// TwinCAT 3 PLC project StageUtils
// Title: StageUtils
// Company: _
// Author: Krystian Lis et al.
// ProjectVersion: 2.0.0
// Description: Various Stage related utilities
// ProgramVersion: 3.1.4026.16
// libraries:
//   Tc2_Standard, * (Beckhoff Automation GmbH)
//   Tc2_System, * (Beckhoff Automation GmbH)
//   StageCore, * (_)
// project tree:
//   Arg/ArgList/ ArgList.TcPOU, I_ArgList.TcIO (not stored), I_MutArgList.TcIO
//   Arg/ArgQueue/ ArgQueue.TcPOU, I_ArgQueue.TcIO, I_MutArgQueue.TcIO
//   Color/ Color.TcDUT, RgbColor.TcPOU
//   Color/Itf/ I_RgbColor.TcIO
//   Entity/CompList/ CompList.TcPOU, I_CompList.TcIO (not stored), I_MutCompList.TcIO
//   Entity/CompSet/ CompSet.TcPOU, I_CompSet.TcIO
//   Math/ Math.TcPOU
//   Time/ GetTaskCycleTime.TcPOU (not stored), GetUnixTime.TcPOU (not stored)
// real-time tasks:
//   TASK Example: cycle T#10ms, priority 20, ADS port 350
//   TASK Test: cycle T#10ms, priority 21, ADS port 351
//   TASK VISU_TASK: cycle T#200000us, priority 30, ADS port 352

// ---- Color/Color.TcDUT
(*
A DWORD alias type to be used with PLC HMI. Encodes RGB value.
*)
TYPE Color : DWORD; END_TYPE

// ---- Arg/ArgList/I_MutArgList.TcIO
(*
A list implementation for managing `I_Arg`.  
*)
INTERFACE I_MutArgList EXTENDS I_ArgList

(*
Adds, updates, or removes an argument in the list at the specified index.  
Return:
- `Ok` - Upon successfully adding, modifying, or removing an entry.
- `Err.Idx` - When attempting to modify an entry at an out-of-bounds index.
*)
METHOD Set : Result
VAR_INPUT
	iIn		: I_Arg;
	nIndex		: UDINT;
END_VAR
END_METHOD

END_INTERFACE

// ---- Arg/ArgQueue/I_ArgQueue.TcIO
(*
A circular queue implementation for managing `I_Arg`.  
*)
INTERFACE I_ArgQueue EXTENDS I_Debug

(*
Returns the current head index of the queue, indicating the next position for insertion.
*)
PROPERTY Head : UDINT
GET
END_GET
END_PROPERTY

PROPERTY Length : UDINT
GET
END_GET
END_PROPERTY

(*
Provides access to the underlying list structure that holds the queue's argument objects.
*)
PROPERTY List : I_ArgList
GET
END_GET
END_PROPERTY

(*
Returns the current tail index of the queue, indicating the next position for retrieval.
*)
PROPERTY Tail : UDINT
GET
END_GET
END_PROPERTY

END_INTERFACE

// ---- Arg/ArgQueue/I_MutArgQueue.TcIO
(*
A circular queue implementation for managing `I_Arg`.  
*)
INTERFACE I_MutArgQueue EXTENDS I_ArgQueue

(*
Clears the queue.
*)
METHOD Clear
END_METHOD

(*
Retrieves and removes the next argument from the queue.  
Advances the tail pointer, ensuring cyclic operation within the queue's capacity.
Returns:
- Ok - Returns `I_Arg`.
- Err.NotFound - Returns null, queue empty.
- Check `I_MutArgList.Get` for more results.
*)
METHOD Pop : Result
VAR_INPUT
	iOut	: REFERENCE TO I_Arg;
END_VAR
END_METHOD

(*
Adds a new argument to the queue.  
Advances the head pointer while maintaining a cyclic structure, and returns an overflow error if the queue is full.
Returns:
- Ok - Successful insertion.
- Err.Ovf - Returns null, the queue is full.
- Check `I_MutArgList.Set` for more results.
*)
METHOD Push : Result
VAR_INPUT
	iIn		: I_Arg;
END_VAR
END_METHOD

END_INTERFACE

// ---- Color/Itf/I_RgbColor.TcIO
(*
Provides methods and properties to operate on RGBA value.
*)
INTERFACE I_RgbColor

(*
ALPHA channel
*)
PROPERTY Alpha : BYTE
GET
END_GET
SET
END_SET
END_PROPERTY

(*
BLUE component
*)
PROPERTY Blue : BYTE
GET
END_GET
SET
END_SET
END_PROPERTY

(*
Clones other components of I_RgbaColor interface.
*)
METHOD Clone
VAR_INPUT
	iColor	: I_RgbColor;
END_VAR
END_METHOD

(*
GREEN component
*)
PROPERTY Green : BYTE
GET
END_GET
SET
END_SET
END_PROPERTY

(*
Compute single Color value from RGBA components when used as getter.
Sets RGBA values by extracting components from a single Color value.
*)
PROPERTY Raw : Color
GET
END_GET
SET
END_SET
END_PROPERTY

(*
RED component
*)
PROPERTY Red : BYTE
GET
END_GET
SET
END_SET
END_PROPERTY

(*
Set each RGBA component value separately.
*)
METHOD Set
VAR_INPUT
	nRed: USINT;
	nGreen: USINT;
	nBlue: USINT;
	nAlpha: USINT;
END_VAR
END_METHOD

END_INTERFACE

// ---- Entity/CompList/I_MutCompList.TcIO
(*
A list implementation for managing `I_Component`.  
*)
INTERFACE I_MutCompList EXTENDS I_CompList

(*
Adds, updates, or removes an argument in the list at the specified index.  
Return:
- `Ok` - Upon successfully adding, modifying, or removing an entry.
- `Err.Idx` - When attempting to modify an entry at an out-of-bounds index.
*)
METHOD Set : Result
VAR_INPUT
	iIn			: I_Component;
	nIndex		: UDINT;
END_VAR
END_METHOD

END_INTERFACE

// ---- Entity/CompSet/I_CompSet.TcIO
INTERFACE I_CompSet

METHOD Append : Result
VAR_INPUT
	iComp: I_Component;
END_VAR
END_METHOD

METHOD Get : Result
VAR_INPUT
	nIdx: UDINT;
	iResult: REFERENCE TO I_Component;
END_VAR
END_METHOD

END_INTERFACE

// ---- Arg/ArgList/ArgList.TcPOU
(*
A list implementation for managing `I_Arg`.  
*)
FUNCTION_BLOCK ArgList
VAR_GENERIC CONSTANT
	nCap	: UDINT := 100;
END_VAR

IMPLEMENTS I_MutArgList

VAR
	_iList	: ARRAY[1..nCap] OF I_Arg;
END_VAR

(*
Provides the maximum capacity of the list.
*)
PROPERTY Cap : UDINT
GET
Cap := nCap;
END_GET
END_PROPERTY

(*
Retrieves the `I_Arg` at the specified index.  
Returns:
- `Ok` - Successfully retrieves the `I_Arg`.
- `Err.Idx` - The specified index is out of bounds.
- `Err.InvRef` - Invalid output reference.
- `Err.Idx` - `iOut` = 0.
*)
METHOD Get : Result
VAR_INPUT
	nIndex		: UDINT;
	iOut		: REFERENCE TO I_Arg;
END_VAR
IF nIndex > nCap OR nIndex = 0 THEN
	Get := Err.Idx;
	RETURN;	
END_IF

IF NOT __ISVALIDREF(iOut) THEN
	Get := Err.InvRef;
	RETURN;
END_IF

iOut := _iList[nIndex];
IF iOut <> 0 THEN
	Get := Ok;
ELSE
	Get := Err.NotFound;
END_IF
END_METHOD

(*
Adds, updates, or removes an argument in the list at the specified index.  
Return:
- `Ok` - Upon successfully adding, modifying, or removing an entry.
- `Err.Idx` - When attempting to modify an entry at an out-of-bounds index.
*)
METHOD Set : Result
VAR_INPUT
	iIn		: I_Arg;
	nIndex		: UDINT;
END_VAR
IF nIndex > nCap OR nIndex = 0 THEN
	Set := Err.Idx;
	RETURN;	
END_IF

_iList[nIndex] := iIn;
Set := Ok;
END_METHOD

END_FUNCTION_BLOCK

// ---- Arg/ArgQueue/ArgQueue.TcPOU
(*
A circular queue implementation for managing `I_Arg`.  
*)
FUNCTION_BLOCK ArgQueue
VAR_GENERIC CONSTANT
	nCap		: UDINT := 100;
END_VAR

IMPLEMENTS I_MutArgQueue

VAR
	_list		: ArgList<nCap>;
	_nLen		: UDINT := 0;
	_nHead		: UDINT := 1;
	_nTail		: UDINT := 1;
END_VAR

(*
Clears the queue.
*)
METHOD Clear
_nHead := 1;
_nTail := 1;
_nLen := 0;
_list.Set(0, 1);
END_METHOD

(*
Returns the current head index of the queue, indicating the next position for insertion.
*)
PROPERTY Head : UDINT
GET
Head := _nHead;
END_GET
END_PROPERTY

PROPERTY Length : UDINT
GET
Length := _nLen;
END_GET
END_PROPERTY

(*
Provides access to the underlying list structure that holds the queue's argument objects.
*)
PROPERTY List : I_ArgList
GET
List := _list;
END_GET
END_PROPERTY

(*
Allows initializing an external interface variable with an interface pointer to this instance within declaration block.
Example:
iQueue: I_MutArgQueue;
queue: ArgQueue := (MutProxy := iQueue);
Result: iQueue <> 0 
*)
PROPERTY MutProxy : REFERENCE TO I_MutArgQueue
SET
MutProxy := THIS^;
END_SET
END_PROPERTY

(*
Retrieves and removes the next argument from the queue.  
Advances the tail pointer, ensuring cyclic operation within the queue's capacity.
Returns:
- Ok - Returns `I_Arg`.
- Err.NotFound - Returns null, queue empty.
- Check `I_ArgList.Get` for more results.
*)
METHOD Pop : Result
VAR_INPUT
	iOut	: REFERENCE TO I_Arg;
END_VAR
IF _nLen = 0 THEN
	Pop := Err.NotFound;
	RETURN;
END_IF;

IF IsOk(_list.Get(_nHead, iOut), nOut => Pop) THEN
	_nHead := (_nHead MOD nCap) + 1;
	_nLen := _nLen - 1;
	Pop := Ok;
END_IF;
END_METHOD

(*
Allows initializing an external interface variable with an interface pointer to this instance within declaration block.
Example:
iQueue: I_ArgQueue;
queue: ArgQueue := (Proxy := iQueue);
Result: iQueue <> 0 
*)
PROPERTY Proxy : REFERENCE TO I_ArgQueue
SET
Proxy := THIS^;
END_SET
END_PROPERTY

(*
Adds a new argument to the queue.  
Advances the head pointer while maintaining a cyclic structure, and returns an overflow error if the queue is full.
Returns:
- Ok - Successful insertion
- Err.Ovf - Returns null, the queue is full.
- Check `I_ArgList.Set` for more results.
*)
METHOD Push : Result
VAR_INPUT
	iIn		: I_Arg;
END_VAR
IF _nLen = nCap THEN
	Push := Err.Ovf;
	RETURN;
END_IF;

IF IsOk(_list.Set(iIn, _nTail), nOut => Push) THEN
	_nTail := (_nTail MOD nCap) + 1;
	_nLen := _nLen + 1;
	Push := Ok;
END_IF;
END_METHOD

(*
Returns the current tail index of the queue, indicating the next position for retrieval.
*)
PROPERTY Tail : UDINT
GET
Tail := _nTail;
END_GET
END_PROPERTY

END_FUNCTION_BLOCK

// ---- Color/RgbColor.TcPOU
(*
Provides methods and properties to operate on RGBA value.
*)
FUNCTION_BLOCK RgbColor IMPLEMENTS I_RgbColor
VAR
	_r: BYTE;
	_g: BYTE;
	_b: BYTE;
	_a: BYTE;
END_VAR

(*
ALPHA channel
*)
PROPERTY Alpha : BYTE
GET
Alpha := _a;
END_GET
SET
_a := Alpha;
END_SET
END_PROPERTY

(*
BLUE component
*)
PROPERTY Blue : BYTE
GET
Blue := _b;
END_GET
SET
_b := Blue;
END_SET
END_PROPERTY

(*
Clones other components of I_RgbaColor interface.
*)
METHOD Clone
VAR_INPUT
	iColor	: I_RgbColor;
END_VAR
IF iColor = 0 THEN
	RETURN;
END_IF

_r := iColor.Red;
_b := iColor.Blue;
_g := iColor.Green;
_a := iColor.Alpha;
END_METHOD

{attribute 'hide'}
METHOD FB_init : BOOL
VAR_INPUT
	bInitRetains : BOOL;
	bInCopyCode : BOOL;
	nRed: USINT;
	nGreen: USINT;
	nBlue: USINT;
	nAlpha: USINT;
END_VAR
Set(nRed, nGreen, nBlue, nAlpha);
END_METHOD

(*
GREEN component
*)
PROPERTY Green : BYTE
GET
Green := _g;
END_GET
SET
_g := Green;
END_SET
END_PROPERTY

(*
Compute single Color value from RGBA components when used as getter.
Sets RGBA values by extracting components from a single Color value.
*)
PROPERTY Raw : Color
GET
Raw := 	USINT_TO_UDINT(_b) OR
			SHL(USINT_TO_UDINT(_g), 8) OR
			SHL(USINT_TO_UDINT(_r), 16) OR
			SHL(USINT_TO_UDINT(_a), 24);
END_GET
SET
_b := UDINT_TO_USINT(Raw AND 16#FF);
_g := UDINT_TO_USINT(SHR(Raw, 8) AND 16#FF);
_r := UDINT_TO_USINT(SHR(Raw, 16) AND 16#FF);
_a := UDINT_TO_USINT(SHR(Raw, 24) AND 16#FF);
END_SET
END_PROPERTY

(*
RED component
*)
PROPERTY Red : BYTE
GET
Red := _r;
END_GET
SET
_r := Red;
END_SET
END_PROPERTY

(*
Set each RGBA component value separately.
*)
METHOD Set
VAR_INPUT
	nRed: USINT;
	nGreen: USINT;
	nBlue: USINT;
	nAlpha: USINT;
END_VAR
_r := nRed;
_g := nGreen;
_b := nBlue;
_a := nAlpha;
END_METHOD

END_FUNCTION_BLOCK

// ---- Entity/CompList/CompList.TcPOU
(*
A list implementation for managing `I_Arg`.  
*)
FUNCTION_BLOCK CompList
VAR_GENERIC CONSTANT
	nCap	: UDINT := 100;
END_VAR

IMPLEMENTS I_MutCompList

VAR
	_iList	: ARRAY[1..nCap] OF I_Component;
END_VAR

(*
Provides the maximum capacity of the list.
*)
PROPERTY Cap : UDINT
GET
Cap := nCap;
END_GET
END_PROPERTY

(*
Retrieves the `I_Component` at the specified index.  
Returns:
- `Ok` - Successfully retrieves the `I_Component`.
- `Err.Idx` - The specified index is out of bounds.
- `Err.InvRef` - Invalid output reference.
- `Err.Idx` - `iOut` = 0.
*)
METHOD Get : Result
VAR_INPUT
	nIndex		: UDINT;
	iOut		: REFERENCE TO I_Component;
END_VAR
IF nIndex > nCap OR nIndex = 0 THEN
	Get := Err.Idx;
	RETURN;	
END_IF

IF NOT __ISVALIDREF(iOut) THEN
	Get := Err.InvRef;
	RETURN;
END_IF

iOut := _iList[nIndex];
IF iOut <> 0 THEN
	Get := Ok;
ELSE
	Get := Err.NotFound;
END_IF
END_METHOD

(*
Adds, updates, or removes an argument in the list at the specified index.  
Return:
- `Ok` - Upon successfully adding, modifying, or removing an entry.
- `Err.Idx` - When attempting to modify an entry at an out-of-bounds index.
*)
METHOD Set : Result
VAR_INPUT
	iIn			: I_Component;
	nIndex		: UDINT;
END_VAR
IF nIndex > nCap OR nIndex = 0 THEN
	Set := Err.Idx;
	RETURN;	
END_IF

_iList[nIndex] := iIn;
Set := Ok;
END_METHOD

END_FUNCTION_BLOCK

// ---- Entity/CompSet/CompSet.TcPOU
FUNCTION_BLOCK CompSet

VAR_GENERIC CONSTANT
	CAP: UDINT := 10;
END_VAR

IMPLEMENTS I_CompSet

VAR_OUTPUT
END_VAR
VAR
	_iComp: ARRAY[1..CAP] OF I_Component;
	_nLen: UDINT;
END_VAR

METHOD Append : Result
VAR_INPUT
	iComp: I_Component;
END_VAR
IF _nLen = CAP THEN
	Append := Err.Ovf;
	RETURN;
END_IF

IF iComp = 0 THEN
	Append := Err.Itf0;
	RETURN;
END_IF

_nLen := _nLen + 1;
_iComp[_nLen] := iComp;
Append := Ok;
END_METHOD

METHOD Get : Result
VAR_INPUT
	nIdx: UDINT;
	iResult: REFERENCE TO I_Component;
END_VAR
IF nIdx = 0 OR nIdx > CAP THEN
	Get := Err.Ovf;
	RETURN;
END_IF

IF NOT __ISVALIDREF(iResult) THEN
	Get := Err.InvRef;
	RETURN;
END_IF

iResult := _iComp[nIdx];
Get := Ok;
END_METHOD

END_FUNCTION_BLOCK

// ---- Math/Math.TcPOU
(*Provides various mathematical functions*)
PROGRAM Math
VAR
END_VAR

(* 
    Time-compensated smoothing coefficient. 
    Alpha = 1 - (1 - B)^dt
*)
METHOD ExptDecay : LREAL
VAR_INPUT
    rBlendFactor : LREAL;   // In [0, 1] — how fast to blend toward input
    rDeltaTime   : LREAL := 0.01;   // In seconds
END_VAR
rBlendFactor := LIMIT(0.0, rBlendFactor, 1.0);
rDeltaTime   := MAX(rDeltaTime, 0.0);
ExptDecay := LIMIT(0.0, 1.0 - EXPT(1.0 - rBlendFactor, rDeltaTime), 1.0);
END_METHOD

(*
First-order low pass filter.
Yt = Xt * Coeff + Y(t-1) * (1- Coeff)
*)
METHOD LowPassFilter : LREAL
VAR_INPUT
	rX				: LREAL;
	rPrvY			: LREAL;
	
	rCoefficient	: LREAL;
END_VAR
LowPassFilter := rX * rCoefficient + rPrvY * (1 - rCoefficient);
END_METHOD

(*
Allows for value normalization with rescalling option.
Returns 0 when rMaxX - rMinX = 0.
*)
METHOD Normalization : LREAL
VAR_INPUT
	rX				: LREAL;
	rMinX			: LREAL;
	rMaxX			: LREAL;
	rMinY			: LREAL := 0;
	rMaxY			: LREAL := 1;
END_VAR
VAR
	_rDnmtr			: LREAL := rMaxX - rMinX;
END_VAR
IF _rDnmtr <> 0 THEN
	Normalization := rMinY + ((rX - rMinX)/_rDnmtr) * (rMaxY - rMinY);
END_IF
END_METHOD

(*
Generates random number every time is called.
*)
METHOD Random : LREAL
VAR_STAT
	_nSeed		: INT;
END_VAR
VAR
	_drand		: Tc2_System.DRAND;
END_VAR
_drand(Seed := _nSeed, Num => Random);
_nSeed := _nSeed + 1;
END_METHOD

END_PROGRAM
